TYPE ST_STATION_Status :
STRUCT

	bSeqIsHoming					: BOOL;
	bStationHomed					:BOOL;		(*FUNCTION Homed*)
	bSeqInProgress				:BOOL;		(*Function In Progress With Cycle*)
	bSeqComplete				:BOOL;		(*Function Complete Cycle - Flag Set After Every Cycle Finsh*)
	bSeqDone					:BOOL;		(*Function Sequence Finished With Success - Flag Set For One PLC Cycle*)
	bStationNotMoving				:BOOL;		(*Function Parts Are Not Moving*)

	bSeqError						: BOOL;
	nSeqErrorID					: UDINT;

END_STRUCT
END_TYPE

(* stored: Version 1.1.0.1, ProductVersion 3.1.4024.15
   DUT ST_STATION_Status: Id {ca4edff0-7187-4a7e-a9d8-347eb908fc88} *)
